{attribute 'global_init_slot' := '49991'}
{attribute 'qualified_only'}
VAR_GLOBAL CONSTANT
	// encoder resolution
	g_incEncoderRes :ARRAY[1..7] OF DINT :=[7(65536)];
	g_absEncoderRes :ARRAY[1..7] OF DINT :=[7(16777216)];
	
	// reduction ratio
	g_motorReduction :ARRAY[1..7] OF LREAL :=[43.9658,26.859,26.8018,(66.0/10)*3,4554.0/130, 4554.0/130,5625.0/361];
	g_absEncoderReduction :ARRAY[1..7] OF LREAL :=[7(1.0)];
	
	// motor parameters
	g_motorTrqConst :ARRAY[1..7] OF LREAL :=[0.0538,0.0538,0.0538,0.0299,0.0193,0.0193,0.0193];
	g_motorMaxCurrent :ARRAY[1..7] OF LREAL :=[1000,1000,1000,1000,300,200,220];//mA
	g_jntMaxTrq :ARRAY[1..7] OF LREAL :=[g_motorMaxCurrent[1]*g_motorReduction[1]*g_motorTrqConst[1]/1000.0,  g_motorMaxCurrent[2]*g_motorReduction[2]*g_motorTrqConst[2]/1000.0,
									g_motorMaxCurrent[3]*g_motorReduction[3]*g_motorTrqConst[3]/1000.0,		g_motorMaxCurrent[4]*g_motorReduction[4]*g_motorTrqConst[4]/1000.0,
									g_motorMaxCurrent[5]*g_motorReduction[5]*g_motorTrqConst[5]/1000.0,		g_motorMaxCurrent[6]*g_motorReduction[6]*g_motorTrqConst[6]/1000.0,
									g_motorMaxCurrent[7]*g_motorReduction[7]*g_motorTrqConst[7]/1000.0];
	
	// motor and absEncoder direction
	g_motorDir :ARRAY[1..2, 1..7] OF INT :=[1, 1, -1, 1, 1, -1, -1,	
											1, 1, -1, 1, 1, -1, -1];
	g_asbEncoderDir :ARRAY[1..2, 1..7] OF INT :=[-1, -1, 1, -1, 1, 1, 1,
												 -1, -1, 1, -1, 1, 1, 1];
																 
	// joint position limit
	//TODO: joint7 is given a large limit for initialization moiton
	//NOTE: joint 4 position is coupled with joint 2/3, so the limit is described by link side
	g_minJntPos: ARRAY[1..2,1..7] OF LREAL:=[-60*g_deg2Rad,	-45*g_deg2Rad-pi/2,		-45*g_deg2Rad, 	-pi/2-220*g_deg2Rad, 	-135*g_deg2Rad+pi,		-45*g_deg2Rad-pi/2,		-330*g_deg2Rad,
											 -60*g_deg2Rad,	-45*g_deg2Rad-pi/2,		-45*g_deg2Rad,	-pi/2+5*g_deg2Rad,		-135*g_deg2Rad+pi,		-45*g_deg2Rad+pi/2,	-330*g_deg2Rad];
	g_maxJntPos: ARRAY[1..2,1..7] OF LREAL:=[60*g_deg2Rad,	60*g_deg2Rad-pi/2,		60*g_deg2Rad,		-pi/2-5*g_deg2Rad,			135*g_deg2Rad+pi,		45*g_deg2Rad-pi/2,		330*g_deg2Rad,
								             60*g_deg2Rad,	60*g_deg2Rad-pi/2,		60*g_deg2Rad,		-pi/2+220*g_deg2Rad,			135*g_deg2Rad+pi,		45*g_deg2Rad+pi/2,		330*g_deg2Rad];
	
	// joint velocity limit
	g_maxJntVel :ARRAY[1..7] OF LREAL :=[7(2*pi)];
	
END_VAR

(* stored: Version 1.1.0.1, ProductVersion 3.1.4024.12
   GVL GVL_ArmJointParameters: Id {cf487053-15bb-46bd-a4ed-bbb1df690beb} *)
